% RSLogix 500 project DIGITALCONTROL.RSS, saved by version 9.00.00.04 %
PROJECT "UNTITLED"    % processor: Bul.1763 MicroLogix 1100 Series B %

PROGRAM FILES
  LAD 2   4 rungs

DATA FILES
  O0 OUTPUT  4 elements
  I1 INPUT  6 elements
  S2 STATUS  66 elements
  B3 BINARY  1 elements
  T4 TIMER  1 elements
  C5 COUNTER  1 elements
  R6 CONTROL  1 elements
  N7 INTEGER  1 elements
  F8 FLOAT  1 elements

LADDER 2
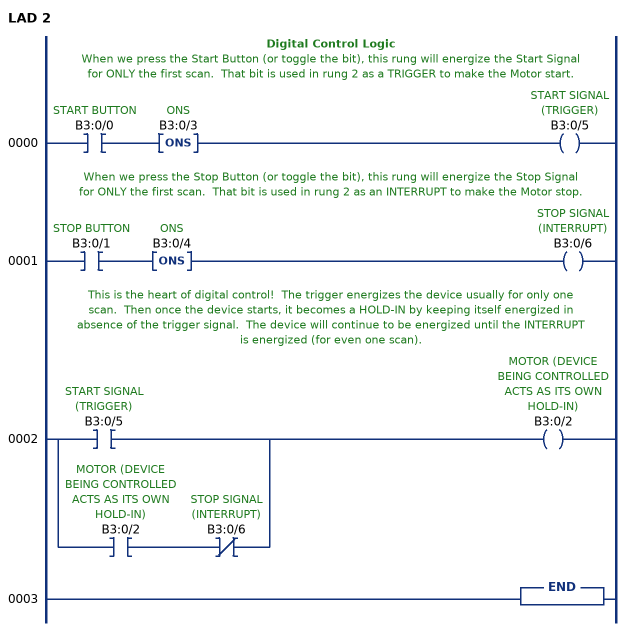
% Rung: 0 %
% TITLE: Digital Control Logic %
% When we press the Start Button (or toggle the bit), this rung will energize the Start Signal for ONLY the first scan.  That bit is used in rung 2 as a TRIGGER to make the Motor start. %
SOR XIC B3:0/0 ONS B3:0/3 OTE B3:0/5 EOR
%   B3:0/0  "START BUTTON" %
%   B3:0/3  "ONS" %
%   B3:0/5  "START SIGNAL (TRIGGER)" %
% Rung: 1 %
% When we press the Stop Button (or toggle the bit), this rung will energize the Stop Signal for ONLY the first scan.  That bit is used in rung 2 as an INTERRUPT to make the Motor stop. %
SOR XIC B3:0/1 ONS B3:0/4 OTE B3:0/6 EOR
%   B3:0/1  "STOP BUTTON" %
%   B3:0/4  "ONS" %
%   B3:0/6  "STOP SIGNAL (INTERRUPT)" %
% Rung: 2 %
% This is the heart of digital control!  The trigger energizes the device usually for only one scan.  Then once the device starts, it becomes a HOLD-IN by keeping itself energized in absence of the trigger signal.  The device will continue to be energized until the INTERRUPT is energized (for even one scan). %
SOR BST XIC B3:0/5 NXB XIC B3:0/2 XIO B3:0/6 BND OTE B3:0/2 EOR
%   B3:0/5  "START SIGNAL (TRIGGER)" %
%   B3:0/2  "MOTOR (DEVICE BEING CONTROLLED ACTS AS ITS OWN HOLD-IN)" %
%   B3:0/6  "STOP SIGNAL (INTERRUPT)" %
% Rung: 3 %
SOR END EOR

OTHER DOCUMENTED ADDRESSES
  N7:0  "VALUE 1"
  N7:1  "LIMIT"
  N7:2  "LIMIT2"
